FUNCTION TryConvert_DINT_TO_STRING : BOOL
VAR_INPUT
	in : DINT;
	out : REFERENCE TO STRING;
END_VAR

out := DINT_TO_STRING(in);
TryConvert_DINT_TO_STRING := TRUE;

END_FUNCTION

(* stored: Version 1.1.0.1, ProductVersion 3.1.4024.12
   POU TryConvert_DINT_TO_STRING: Id {bcf1e215-4387-4906-9ba7-0727fa6126c6}, SpecialFunc None *)
